// TwinCAT 3 PLC project MAS418_PLC
// ProgramVersion: 3.1.4023.0
// libraries:
//   Tc2_Standard, * (Beckhoff Automation GmbH)
//   Tc2_System, * (Beckhoff Automation GmbH)
//   Tc3_Module, * (Beckhoff Automation GmbH)
// project tree:
//   / GlobalTextList.TcGTLO, PlcTask.TcTTO, Visualization Manager.TcVMO (not stored)
//   POUs/ MAIN.TcPOU
//   VISUs/ HMI.TcVIS

CONFIGURATION MAS418_PLC
    RESOURCE PLC ON TwinCAT3
        TASK PlcTask(INTERVAL := T#10ms, PRIORITY := 20);
        PROGRAM MAIN WITH PlcTask : MAIN;
    END_RESOURCE
END_CONFIGURATION

// ---- POUs/MAIN.TcPOU
PROGRAM MAIN
VAR
	bEnable : BOOL;
	bStart : BOOL;
	nINT : INT := -32768;
	nUINT : UINT := 65535;
	fREAL : REAL := 255.255;
	nFloatConversion : INT;
	fFloatConversion : LREAL;
	nIntConversion : INT;
	fIntConversion : LREAL;
	

	
END_VAR

bEnable := bStart;
fFloatConversion := INT_TO_LREAL(nFloatConversion);
nIntConversion := LREAL_TO_INT(fIntConversion);

END_PROGRAM

// ---- GlobalTextList.TcGTLO
TEXTLIST GlobalTextList
  731 = '%f'
  446 = '%i'
  512 = '%s'
  280 = 'BOOL'
  402 = 'DataTypeTesting'
  906 = 'INT'
  802 = 'light'
  361 = 'Power ON'
  281 = 'Powerswitch'
  798 = 'REAL'
  657 = 'STRING'
  709 = 'UINT'
  858 = 'UINY'
END_TEXTLIST

// ---- VISUs/HMI.TcVIS
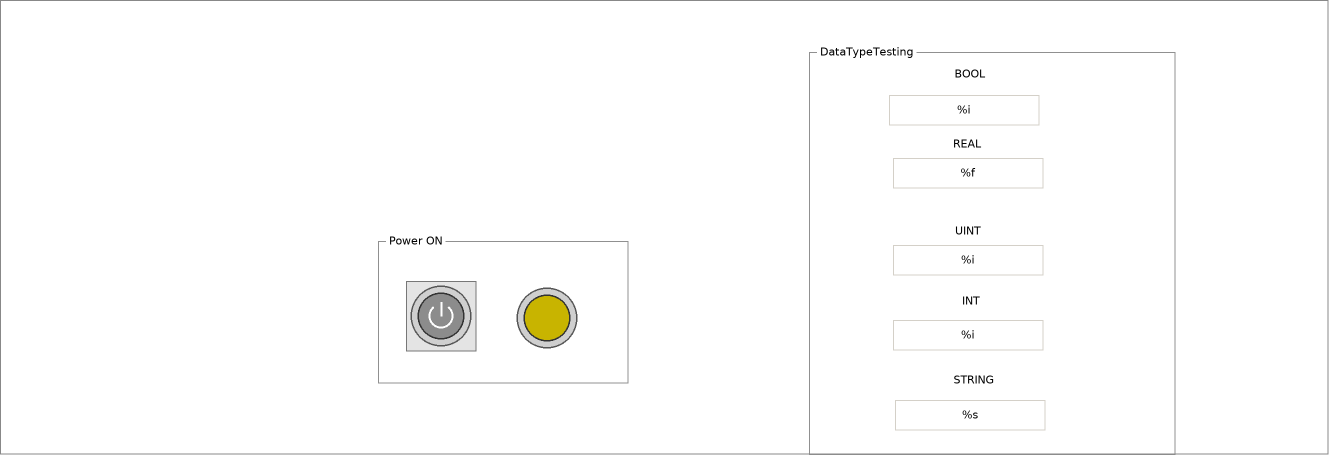
VISUALIZATION HMI  // 1329x455
    GroupBox (378,233 250x150), "Power ON"
        PowerSwitch (28,48 70x70), tooltip "Powerswitch", variable: MAIN.bStart, behaviour: TOGGLE, style: Switch-PowerSwitch-Gray
        Lamp1 (134,50 70x70), tooltip "light", variable: MAIN.bEnable, style: Lamp-Lamp1-Yellow
    GroupBox (809,44 366x411), "DataTypeTesting"
        Textfield (80,51 150x30), "%i", text variable: MAIN.nINT
        Textfield (84,114 150x30), "%f", text variable: MAIN.fREAL
        Textfield (84,276 150x30), "%i"
        Textfield (86,356 150x30), "%s"
        Textfield (84,201 150x30), "%i", text variable: MAIN.nUINT
        Label (86,15 150x30), "BOOL"
        Label (83,85 150x30), "REAL"
        Label (84,172 150x30), "UINT"
        Label (87,242 150x30), "INT"
        Label (90,321 150x30), "STRING"
    Label (1179,249 150x30)
END_VISUALIZATION
